// TIA Portal project "Uklad_3_rzedu_OPC_comm" (V16)

(* hardware
DEVICE "S71500/ET200MP station_1"  S7-1500 station
   slot 0: "Rail_0"  Rack  6ES7 590-1***0-0AA0
   slot 1: "PLCMatlabOPCUA"  CPU 1511-1 PN  6ES7 511-1AK02-0AB0  V2.6
      slot 3: "CPU display_1"  6ES7591-1AA00-0AA0
      slot 32768: "PROFINET interface_1"  X1
DEVICE "HMI_PLCSIM_Adv"  TP1200 Comfort
   slot 0: "TP1200 Comfort"  TP1200 Comfort  6AV2 124-0MC01-0AX0  14.0.0.0
   slot 1: "HMI_RT_3"  TP1200 Comfort  6AV2 124-0MC01-0AX0  14.0.0.0
   slot 5: "HMI_PLCSim.IE_CP_1"  PROFINET Interface  14.0.0.0
      slot 1: "PROFINET Interface_1"  PROFINET Interface
         slot 1: "Port_1"  Port
         slot 2: "Port_2"  Port
   slot 7: "HMI_PLCSim.MPI/DP_CP_1"  MPI/DP Interface  14.0.0.0
*)

// ===== PLC "PLCMatlabOPCUA"  CPU 1511-1 PN =====

VAR_GLOBAL   // PLC tag table "Default tag table"
   "inputAngleSFunc" AT %I0.0 : LReal;
   "outputForceSFunc" AT %Q0.0 : LReal;
END_VAR

DATA_BLOCK "MatlabData"   // DB6
{ S7_Optimized_Access := 'TRUE' }
VERSION : 0.1
   VAR
      rSetLevelSquareTank : Real;   // wartosc zadana poziomu w kwadrotowym zbiorniku
      lrActLevelSquareTank : LReal;   // wartosc aktualna poziomu w kwadrotowym zbiorniku
      rSetLevelTrapzezoidTank : Real;   // wartosc zadana poziomu w trapezowym zbiorniku
      lrActLevelTrapzezoidTank : LReal;   // wartosc aktualna poziomu w trapezowym zbiorniku
      rSetLevelRoundTank : Real;   // wartosc zadana poziomu w okraglym zbiorniku
      lrActLevelRoundTank : LReal;   // wartosc aktualna poziomu w okraglym zbiorniku
   END_VAR
BEGIN
END_DATA_BLOCK

DATA_BLOCK "Tanks"   // DB13
{ S7_Optimized_Access := 'TRUE' }
VERSION : 0.1
   VAR
      SquareTankData : Struct
         iSetpoint : Int := 0;
         iManualOutputPercentage : Int := 0;   // %
         xManualOutputEnable : Bool;
         iOperatingMode : Int := 3;
      END_STRUCT;
      TrapezoidTankData : Struct
         iSetpoint : Int := 0;
         iManualOutputPercentage : Int := 0;   // %
         xManualOutputEnable : Bool;
         iOperatingMode : Int := 3;
      END_STRUCT;
      RoundTankData : Struct
         iSetpoint : Int := 0;
         iManualOutputPercentage : Int := 0;   // %
         xManualOutputEnable : Bool;
         iOperatingMode : Int := 3;
      END_STRUCT;
      SquareTankActivation : Bool;
      TrapezoidTankActivation : Bool;
      RoundTankActivation : Bool;
      testbit : Bool;
   END_VAR
BEGIN
END_DATA_BLOCK

ORGANIZATION_BLOCK "Main"   // OB1, LAD, ProgramCycle
TITLE = "Main Program Sweep (Cycle)"
{ S7_Optimized_Access := 'TRUE' }
VERSION : 0.1
   VAR_INPUT
      Initial_Call : Bool;   // Initial call of this OB
      Remanence : Bool;   // =True, if remanent data are available
   END_VAR
BEGIN
END_ORGANIZATION_BLOCK

ORGANIZATION_BLOCK "Cyclic20ms"   // OB30, SCL, CyclicInterrupt
{ S7_Optimized_Access := 'TRUE' }
VERSION : 0.1
   VAR_INPUT
      Initial_Call : Bool;   // Initial call of this OB
      Event_Count : Int;   // Events discarded
   END_VAR
   VAR_TEMP
      tempOutputPercentage : Real;
   END_VAR
BEGIN

   REGION PIDs

       IF "Tanks".SquareTankActivation THEN

           "InstPID_SquareTank"(Setpoint := "Tanks".SquareTankData.iSetpoint,
                                Input := LREAL_TO_REAL("MatlabData".lrActLevelSquareTank),
                                ManualEnable := "Tanks".SquareTankData.xManualOutputEnable,
                                ManualValue := "Tanks".SquareTankData.iManualOutputPercentage,
                                ModeActivate := TRUE,
                                Output => "MatlabData".rSetLevelSquareTank,
                                Mode := "Tanks".SquareTankData.iOperatingMode);

       ELSIF "Tanks".TrapezoidTankActivation THEN

           "InstPID_TrapzezoidTank"(Setpoint := "Tanks".TrapezoidTankData.iSetpoint,
                                    Input := LREAL_TO_REAL("MatlabData".lrActLevelTrapzezoidTank),
                                    ManualEnable := "Tanks".TrapezoidTankData.xManualOutputEnable,
                                    ManualValue := "Tanks".TrapezoidTankData.iManualOutputPercentage,
                                    ModeActivate := TRUE,
                                    Output => "MatlabData".rSetLevelSquareTank,
                                    Mode := "Tanks".TrapezoidTankData.iOperatingMode);

       ELSIF "Tanks".RoundTankActivation THEN

           "InstPID_RoundTank"(Setpoint := "Tanks".RoundTankData.iSetpoint,
                               Input := LREAL_TO_REAL("MatlabData".lrActLevelRoundTank),
                               ManualEnable := "Tanks".RoundTankData.xManualOutputEnable,
                               ManualValue := "Tanks".RoundTankData.iManualOutputPercentage,
                               ModeActivate := TRUE,
                               Output => "MatlabData".rSetLevelSquareTank,
                               Mode := "Tanks".RoundTankData.iOperatingMode);
       ELSE
           "MatlabData".rSetLevelSquareTank := 0;
       END_IF;

   END_REGION
END_ORGANIZATION_BLOCK

(* ===== HMI "HMI_RT_3" =====
system functions are stored by id; their names below are inferred from use
connection "HMI_Connection_PLCSim": ETHERNET, S7_1500_OMS

HMI tags "Default tag table"
   "SquareTankData.iManualOutputPercentage" : Int = PLC Tanks.SquareTankData.iManualOutputPercentage, 100 ms
   "SquareTankData.xManualOutputEnable" : Bool = PLC Tanks.SquareTankData.xManualOutputEnable, 100 ms
   "SquareTankData.iOperatingMode" : Int = PLC Tanks.SquareTankData.iOperatingMode, 100 ms
   "lrActLevelSquare" : LReal = PLC MatlabData.lrActLevelSquareTank, 100 ms
   "SquareTankData.iSetpoint" : Int = PLC Tanks.SquareTankData.iSetpoint, 100 ms
   "rSetLevelSquare" : Real = PLC MatlabData.rSetLevelSquareTank, 100 ms
   "Tanks.SquareTankActivation" : Bool = PLC Tanks.SquareTankActivation, 1 s
   "Tanks.TrapezoidTankActivation" : Bool = PLC Tanks.TrapezoidTankActivation, 1 s
   "Tanks.RoundTankActivation" : Bool = PLC Tanks.RoundTankActivation, 1 s
   "Tanks.TrapezoidTankData.iSetpoint" : Int = PLC Tanks.TrapezoidTankData.iSetpoint, 1 s
   "MatlabData.lrActLevelTrapzezoidTank" : LReal = PLC MatlabData.lrActLevelTrapzezoidTank, 1 s
   "Tanks.TrapezoidTankData.xManualOutputEnable" : Bool = PLC Tanks.TrapezoidTankData.xManualOutputEnable, 1 s
   "Tanks.TrapezoidTankData.iManualOutputPercentage" : Int = PLC Tanks.TrapezoidTankData.iManualOutputPercentage, 1 s
   "Tanks.RoundTankData.iSetpoint" : Int = PLC Tanks.RoundTankData.iSetpoint, 1 s
   "MatlabData.lrActLevelRoundTank" : LReal = PLC MatlabData.lrActLevelRoundTank, 1 s
   "Tanks.RoundTankData.iManualOutputPercentage" : Int = PLC Tanks.RoundTankData.iManualOutputPercentage, 1 s
   "Tanks.RoundTankData.xManualOutputEnable" : Bool = PLC Tanks.RoundTankData.xManualOutputEnable, 1 s
   "MatlabData.rSetLevelTrapzezoidTank" : Real = PLC MatlabData.rSetLevelTrapzezoidTank, 1 s
   "MatlabData.rSetLevelRoundTank" : Real = PLC MatlabData.rSetLevelRoundTank, 1 s

text list "ManualEnable": 0 'AUTO'; 1 'MANUAL'

text list "Text_list_2": 0 'KWADRATOWY'; 1 'KWADRATOWY'

text list "Text_list_1": 0..1 'TRAPEZ'

text list "Text_list_3": 0..1 'OKRĄGŁY'

text list "ManualEnable_2": 0 'AUTO'; 1 'MANUAL'

text list "ManualEnable_1": 0 'AUTO'; 1 'MANUAL'

screen "Visu_Tanks_Control" 1280x800
   TrendView "Trendview" at 316,10 size 953x779
      Visibility <- "Tanks.SquareTankActivation"
   IOField "CurrenAngle" at 180,83 size 113x24; FormatPattern s9999.999
      ProcessValue <- "lrActLevelSquare"
   IOField "Setpoint" at 180,55 size 113x24; FormatPattern s999
      ProcessValue <- "SquareTankData.iSetpoint"
   Slider "ManualOutput" at 20,157 size 280x48; Caption 'SIMATIC'
      ProcessValue <- "SquareTankData.iManualOutputPercentage"
   Button "Manual Override" at 20,117 size 280x32; TextOff 'AUTO'; TextOn 'MANUAL'; TextList "ManualEnable"
      on Click: InvertBit("SquareTankData.xManualOutputEnable")
      Appearance <- "SquareTankData.xManualOutputEnable"
      ProcessValue <- "SquareTankData.xManualOutputEnable"
   TextField "Text field_2" at 20,55 size 112x22; Text 'POZIOM ZAD'
   TextField "Text field_3" at 20,79 size 111x22; Text 'POZIOM AKT'
   Button "Button_1" at 69,20 size 185x28; TextOff 'KWADRAT OFF'; TextOn 'KWADRAT ON'; TextList "Text_list_2"
      on Click: InvertBit("Tanks.SquareTankActivation"); ResetBit("Tanks.TrapezoidTankActivation"); ResetBit("Tanks.RoundTankActivation")
      Appearance <- "Tanks.SquareTankActivation"
      ProcessValue <- "Tanks.SquareTankActivation"
   IOField "CurrenAngle_1" at 181,344 size 113x24; FormatPattern s9999.999
      ProcessValue <- "MatlabData.lrActLevelTrapzezoidTank"
   IOField "Setpoint_1" at 181,316 size 113x24; FormatPattern s999
      ProcessValue <- "Tanks.TrapezoidTankData.iSetpoint"
   Slider "ManualOutput_1" at 21,418 size 280x48; Caption 'SIMATIC'
      ProcessValue <- "Tanks.TrapezoidTankData.iManualOutputPercentage"
   Button "Manual Override_1" at 21,378 size 280x32; TextOn 'MANUAL'; TextOff 'AUTO'; TextList "ManualEnable_1"
      on Click: InvertBit("Tanks.TrapezoidTankData.xManualOutputEnable")
      ProcessValue <- "Tanks.TrapezoidTankData.xManualOutputEnable"
      Appearance <- "Tanks.TrapezoidTankData.xManualOutputEnable"
   TextField "Text field_1" at 21,316 size 112x22; Text 'POZIOM ZAD'
   TextField "Text field_4" at 21,340 size 111x22; Text 'POZIOM AKT'
   IOField "CurrenAngle_2" at 180,611 size 113x24; FormatPattern s9999.999
      ProcessValue <- "MatlabData.lrActLevelRoundTank"
   IOField "Setpoint_2" at 180,583 size 113x24; FormatPattern s999
      ProcessValue <- "Tanks.RoundTankData.iSetpoint"
   Slider "ManualOutput_2" at 20,685 size 280x48; Caption 'SIMATIC'
      ProcessValue <- "Tanks.RoundTankData.iManualOutputPercentage"
   Button "Manual Override_2" at 20,645 size 280x32; TextOn 'MANUAL'; TextOff 'AUTO'; TextList "ManualEnable_2"
      on Click: InvertBit("Tanks.RoundTankData.xManualOutputEnable")
      ProcessValue <- "Tanks.RoundTankData.xManualOutputEnable"
      Appearance <- "Tanks.RoundTankData.xManualOutputEnable"
   TextField "Text field_5" at 20,583 size 112x22; Text 'POZIOM ZAD'
   TextField "Text field_6" at 20,607 size 111x22; Text 'POZIOM AKT'
   Button "Button_2" at 69,278 size 185x32; TextOn 'KWADRAT ON'; TextOff 'KWADRAT OFF'; TextList "Text_list_1"
      on Click: InvertBit("Tanks.TrapezoidTankActivation"); ResetBit("Tanks.RoundTankActivation"); ResetBit("Tanks.SquareTankActivation")
      ProcessValue <- "Tanks.TrapezoidTankActivation"
      Appearance <- "Tanks.TrapezoidTankActivation"
   Button "Button_3" at 69,543 size 185x32; TextOn 'KWADRAT ON'; TextOff 'KWADRAT OFF'; TextList "Text_list_3"
      on Click: InvertBit("Tanks.RoundTankActivation"); ResetBit("Tanks.SquareTankActivation"); ResetBit("Tanks.TrapezoidTankActivation")
      ProcessValue <- "Tanks.RoundTankActivation"
      Appearance <- "Tanks.RoundTankActivation"
   TrendView "Trendview_1" at 311,9 size 953x779
      Visibility <- "Tanks.TrapezoidTankActivation"
   TrendView "Trendview_2" at 310,10 size 953x779
      Visibility <- "Tanks.RoundTankActivation"
*)